{attribute 'reflection'}
FUNCTION_BLOCK T_Notification IMPLEMENTS I_Notification
VAR
    EventHandlers : T_ListONotificationHandlers(Capacity := 5);
    _Args : T_Stream(StreamLength := 8);
END_VAR

METHOD AddNotificationHandler : I_Notification
VAR_INPUT
    Handler : I_NotificationHandler;
END_VAR
EventHandlers.AddHandler(Handler);
AddNotificationHandler := THIS^;
END_METHOD

PROPERTY PUBLIC Args : I_StreamWriter
GET
Args := _Args;
END_GET
END_PROPERTY

METHOD ClearNotificationHandlers : I_Notification
EventHandlers.Clear();
ClearNotificationHandlers := THIS^;
END_METHOD

METHOD Raise
VAR
    Handler : I_NotificationHandler;
    i : UDINT;
END_VAR
IF EventHandlers.Count > 0 THEN
    FOR i := 0 TO EventHandlers.Count - 1 DO
        Handler := EventHandlers.GetHandler(i);
        IF Handler <> 0 THEN
            _Args.Seek(0); // to ensure that each handler reads args from start of the stream
            Handler.OnNotificationReceived(Args := _Args);
        END_IF
    END_FOR
END_IF
_Args.Clear(); // to leave event args empty for next time event is raised
END_METHOD

END_FUNCTION_BLOCK

(* stored: Version 1.1.0.1, ProductVersion 3.1.4024.6
   POU T_Notification: Id {34c3e11c-b24b-47fd-988a-f99b18a3f2ec}, SpecialFunc None
   Folder Methods: Id {b30ccf79-62ad-46da-a613-c3db6aa14265}
   Folder Properties: Id {376ef0d4-0330-4112-ac16-061d4f2c6035}
   Method AddNotificationHandler: Id {bad47bb4-23ca-4961-a375-b50fdcef3f1a}
   Property Args: Id {81d2c015-f4cb-4582-8ade-a9757b20d5f0}
   Get Get: Id {74639c3f-ebbc-4092-a1f0-5bf037d256a8}
   Method ClearNotificationHandlers: Id {505e6c2b-db1c-4664-9c9e-5c68fcd6cf2b}
   Method Raise: Id {96b98869-baef-4dec-8667-b534757ed3a1} *)
